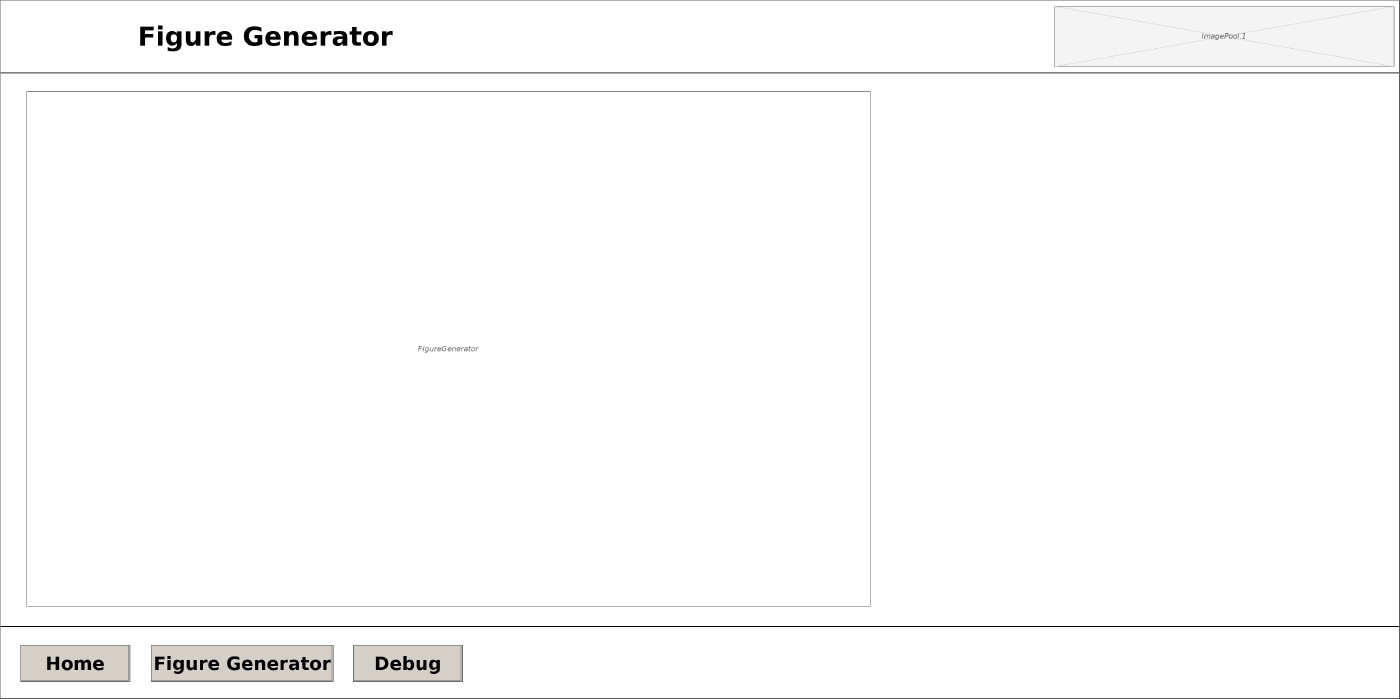
VISUALIZATION FigureGenerator1  // 1919x959
    Rectangle (0,0 1919x910)
    Rectangle (0,0 1919x100)
    Rectangle (0,859 1919x100)
    Button (28,885 150x50), "Home"
        OnMouseClick: change screen: Home
    Label (193,25 342x50), "Figure Generator"
    Image (1445,8 466x83), image: ImagePool.1
    Button (207,885 250x50), "Figure Generator"
    Button (484,885 150x50), "Debug"
        OnMouseClick: change screen: Debug
    Frame (36,125 1157x707)
        shows FigureGenerator()
END_VISUALIZATION

(* stored: Version 1.1.0.1, ProductVersion 3.1.4024.12
   Visu FigureGenerator1: Id {a506a3c8-c118-410e-a7dc-977b70adf055} *)
